FUNCTION_BLOCK FB_HeavyWash IMPLEMENTS I_WashStrategy
VAR
	
	nRinseCount : INT := 1;
	iMotorRef : I_Motor;
	bWashing : BOOL;
	bDrying : BOOL;
	
	tWashTime : TIME := T#20S;
	nMotorWashSpeed : INT := 300;
	
	nMotorDrySpeed : INT := 1000; 
	nMotorDryTime : TIME := T#15S;
	
	fbWashTimer : TON;
END_VAR

{warning 'add method implementation '}
METHOD GetDuration : TIME
VAR
END_VAR
GetDuration := tWashTime * (nRinseCount+1) + nMotorDryTime ;
END_METHOD

METHOD GetRinseCount : INT
VAR_INPUT
END_VAR
GetRinseCount := nRinseCount+1;
END_METHOD

METHOD StartSpin : BOOL
VAR_INPUT
END_VAR
bDrying := TRUE;
fbWashTimer( IN := bDrying, PT := nMotorDryTime);
IF NOT fbWashTimer.Q THEN
	iMotorRef.DrySpin(nMotorDrySpeed);
ELSE
	iMotorRef.Stop();
	bDrying := FALSE;
	fbWashTimer( IN := bDrying);
	StartSpin := TRUE;
END_IF
END_METHOD

{warning 'add method implementation '}
METHOD StartWash : BOOL
VAR_INPUT
	iMotor : I_Motor;
END_VAR
iMotorRef := iMotor;
bWashing := TRUE;
fbWashTimer( IN := bWashing, PT := tWashTime);
IF NOT fbWashTimer.Q THEN
	iMotorRef.WashSpin(nMotorWashSpeed);
ELSE
	iMotorRef.Stop();
	bWashing := FALSE;
	fbWashTimer( IN := bWashing);
	StartWash := TRUE;
END_IF
END_METHOD

{warning 'add method implementation '}
METHOD Stop
bWashing := FALSE;
END_METHOD

END_FUNCTION_BLOCK

(* stored: Version 1.1.0.1, ProductVersion 3.1.4024.16
   POU FB_HeavyWash: Id {9f802e7e-d184-4f69-9a2e-1ffb9c72b5ed}, SpecialFunc None
   Method GetDuration: Id {6be335db-62b9-48ff-8041-697cb1ae4e21}
   Method GetRinseCount: Id {8bba1237-230e-4279-8dfc-e7cf947fc9e1}
   Method StartSpin: Id {d2b8b77a-30a9-49ed-8f32-df6f051eabaf}
   Method StartWash: Id {27fd2ba4-aad3-4a3c-aa84-7dce93d77d83}
   Method Stop: Id {95f3ec6f-32e8-476b-97eb-56e90e6958cc} *)
